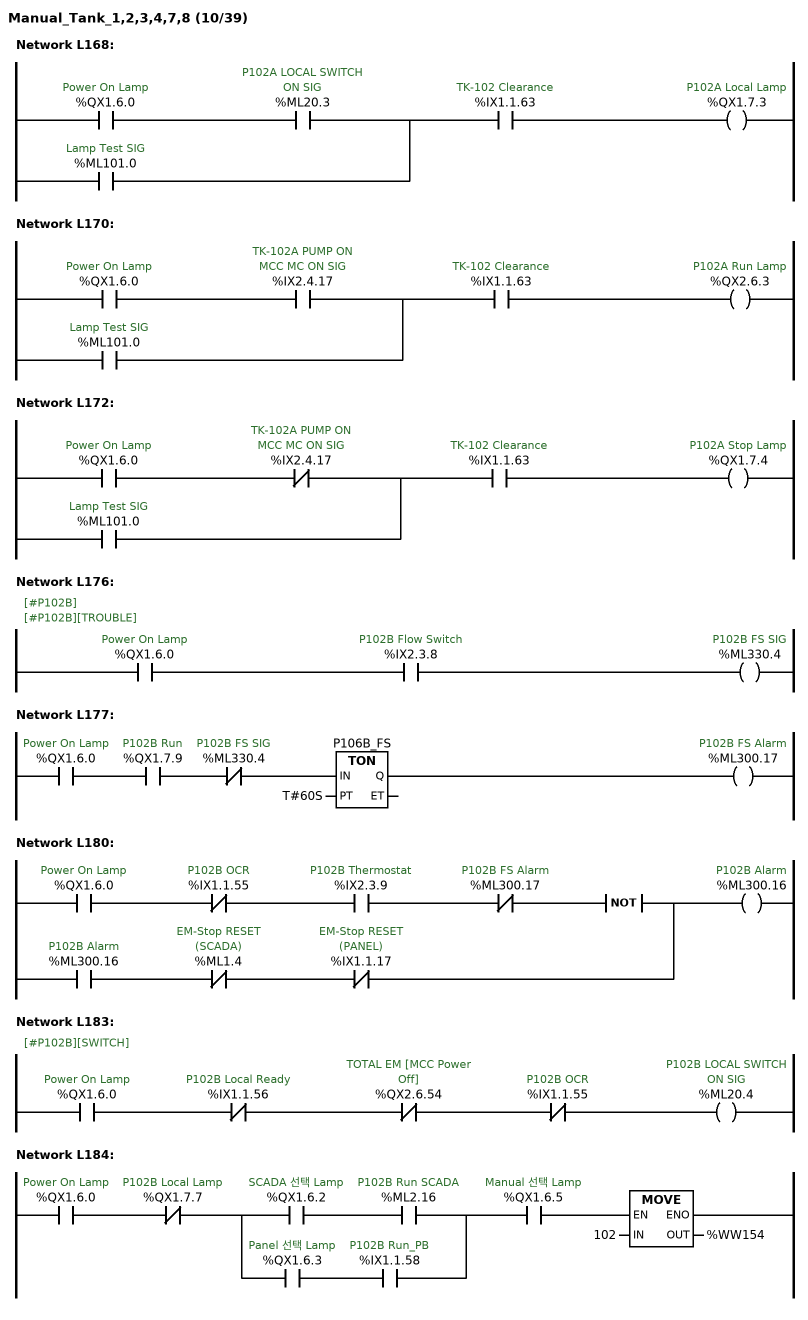
(* [picture p24: Manual_Tank_1,2,3,4,7,8 rungs L168-L184] *)
(* Rung L168 *)
%QX1.7.3 := ((%QX1.6.0 AND %ML20.3) OR %ML101.0) AND %IX1.1.63;
(* Rung L170 *)
%QX2.6.3 := ((%QX1.6.0 AND %IX2.4.17) OR %ML101.0) AND %IX1.1.63;
(* Rung L172 *)
%QX1.7.4 := ((%QX1.6.0 AND NOT %IX2.4.17) OR %ML101.0) AND %IX1.1.63;
(* [#P102B] *)
(* [#P102B][TROUBLE] *)
(* Rung L176 *)
%ML330.4 := %QX1.6.0 AND %IX2.3.8;
(* Rung L177 *)
P106B_FS(IN := %QX1.6.0 AND %QX1.7.9 AND NOT %ML330.4, PT := T#60S);
%ML300.17 := P106B_FS.Q;
(* Rung L180 *)
%ML300.16 := NOT (%QX1.6.0 AND NOT %IX1.1.55 AND %IX2.3.9 AND NOT %ML300.17) OR (%ML300.16 AND NOT %ML1.4 AND NOT %IX1.1.17);
(* [#P102B][SWITCH] *)
(* Rung L183 *)
%ML20.4 := %QX1.6.0 AND NOT %IX1.1.56 AND NOT %QX2.6.54 AND NOT %IX1.1.55;
(* Rung L184 *)
IF %QX1.6.0 AND NOT %QX1.7.7 AND ((%QX1.6.2 AND %ML2.16) OR (%QX1.6.3 AND %IX1.1.58)) AND %QX1.6.5 THEN
    %WW154 := 102;
END_IF;

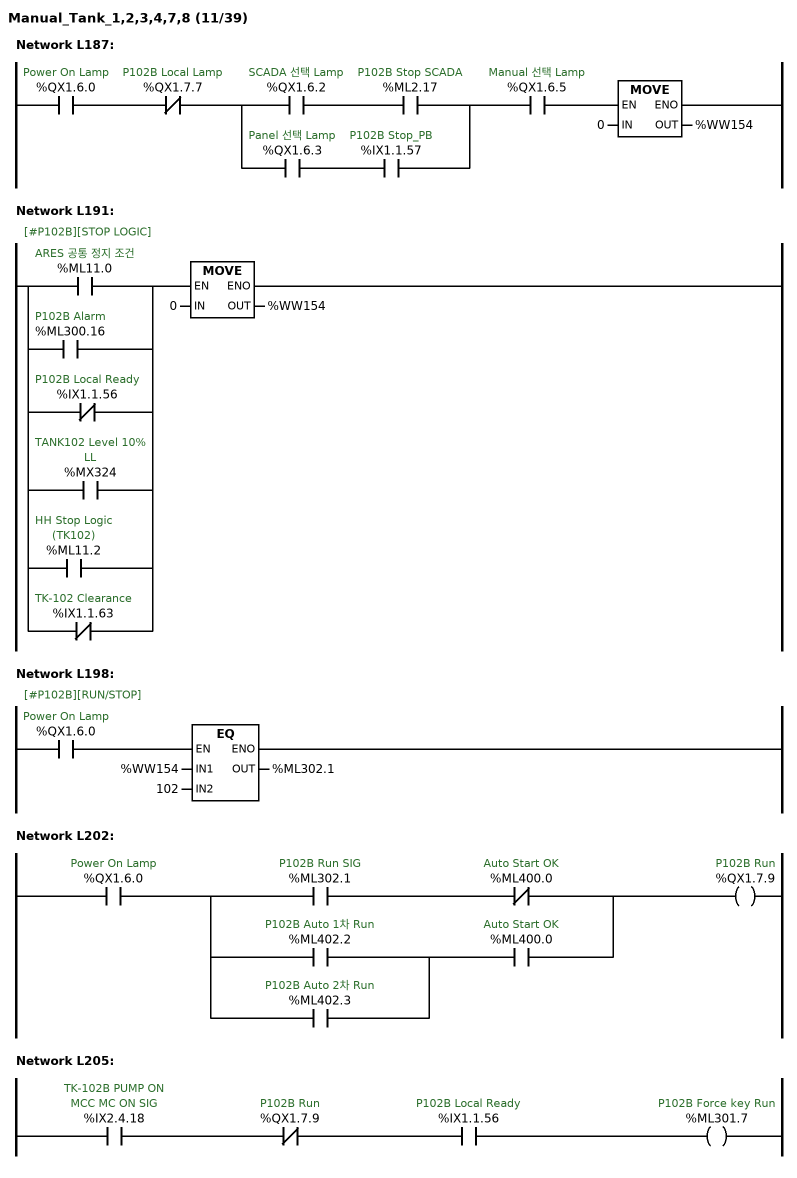
(* Rung L187 *)
IF %QX1.6.0 AND NOT %QX1.7.7 AND ((%QX1.6.2 AND %ML2.17) OR (%QX1.6.3 AND %IX1.1.57)) AND %QX1.6.5 THEN
    %WW154 := 0;
END_IF;
(* [#P102B][STOP LOGIC] *)
(* Rung L191 *)
IF %ML11.0 OR %ML300.16 OR NOT %IX1.1.56 OR %MX324 OR %ML11.2 OR NOT %IX1.1.63 THEN %WW154 := 0; END_IF;
(* [#P102B][RUN/STOP] *)
(* Rung L198 *)
IF %QX1.6.0 THEN %ML302.1 := %WW154 = 102; END_IF;
(* Rung L202 *)
%QX1.7.9 := %QX1.6.0 AND ((%ML302.1 AND NOT %ML400.0) OR ((%ML402.2 OR %ML402.3) AND %ML400.0));
(* Rung L205 *)
%ML301.7 := %IX2.4.18 AND NOT %QX1.7.9 AND %IX1.1.56;

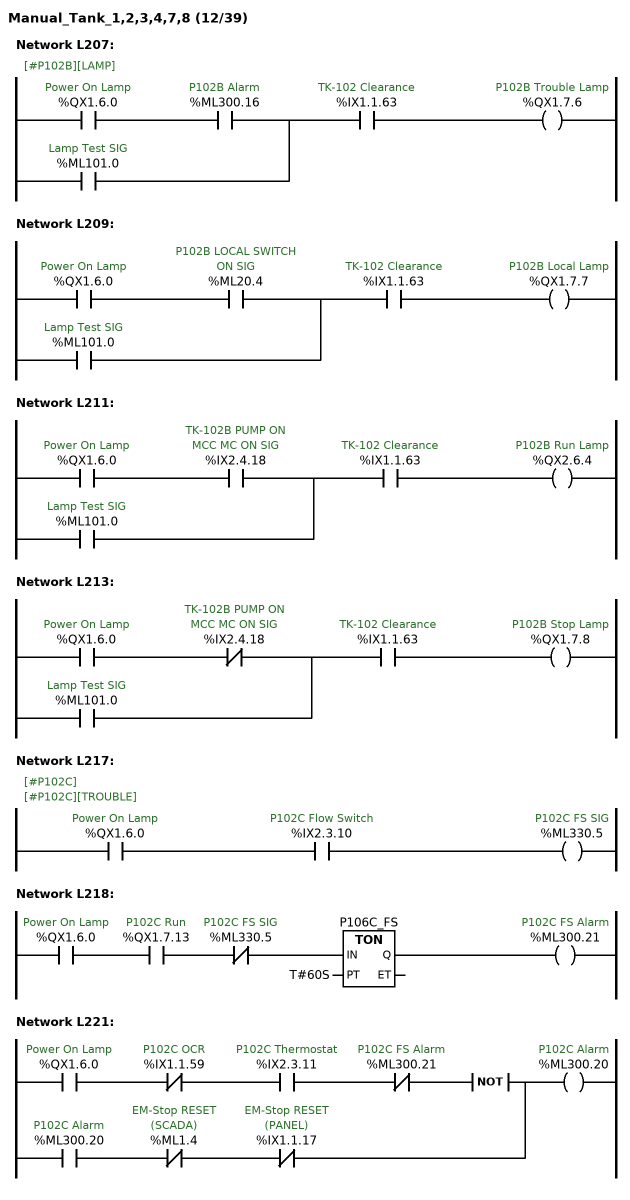
(* [#P102B][LAMP] *)
(* Rung L207 *)
%QX1.7.6 := ((%QX1.6.0 AND %ML300.16) OR %ML101.0) AND %IX1.1.63;
(* Rung L209 *)
%QX1.7.7 := ((%QX1.6.0 AND %ML20.4) OR %ML101.0) AND %IX1.1.63;
(* Rung L211 *)
%QX2.6.4 := ((%QX1.6.0 AND %IX2.4.18) OR %ML101.0) AND %IX1.1.63;
(* Rung L213 *)
%QX1.7.8 := ((%QX1.6.0 AND NOT %IX2.4.18) OR %ML101.0) AND %IX1.1.63;
(* [#P102C] *)
(* [#P102C][TROUBLE] *)
(* Rung L217 *)
%ML330.5 := %QX1.6.0 AND %IX2.3.10;
(* Rung L218 *)
P106C_FS(IN := %QX1.6.0 AND %QX1.7.13 AND NOT %ML330.5, PT := T#60S);
%ML300.21 := P106C_FS.Q;
(* Rung L221 *)
%ML300.20 := NOT (%QX1.6.0 AND NOT %IX1.1.59 AND %IX2.3.11 AND NOT %ML300.21) OR (%ML300.20 AND NOT %ML1.4 AND NOT %IX1.1.17);

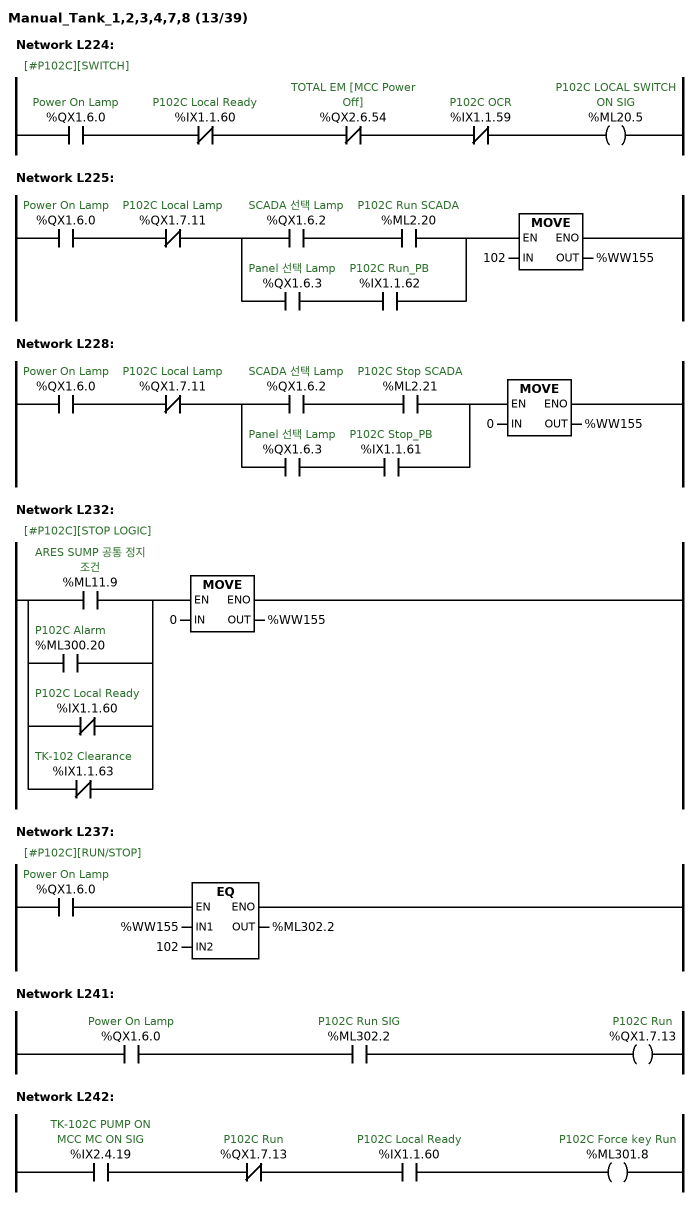
(* [#P102C][SWITCH] *)
(* Rung L224 *)
%ML20.5 := %QX1.6.0 AND NOT %IX1.1.60 AND NOT %QX2.6.54 AND NOT %IX1.1.59;
(* Rung L225 *)
IF %QX1.6.0 AND NOT %QX1.7.11 AND ((%QX1.6.2 AND %ML2.20) OR (%QX1.6.3 AND %IX1.1.62)) THEN
    %WW155 := 102;
END_IF;
(* Rung L228 *)
IF %QX1.6.0 AND NOT %QX1.7.11 AND ((%QX1.6.2 AND %ML2.21) OR (%QX1.6.3 AND %IX1.1.61)) THEN
    %WW155 := 0;
END_IF;
(* [#P102C][STOP LOGIC] *)
(* Rung L232 *)
IF %ML11.9 OR %ML300.20 OR NOT %IX1.1.60 OR NOT %IX1.1.63 THEN %WW155 := 0; END_IF;
(* [#P102C][RUN/STOP] *)
(* Rung L237 *)
IF %QX1.6.0 THEN %ML302.2 := %WW155 = 102; END_IF;
(* Rung L241 *)
%QX1.7.13 := %QX1.6.0 AND %ML302.2;
(* Rung L242 *)
%ML301.8 := %IX2.4.19 AND NOT %QX1.7.13 AND %IX1.1.60;

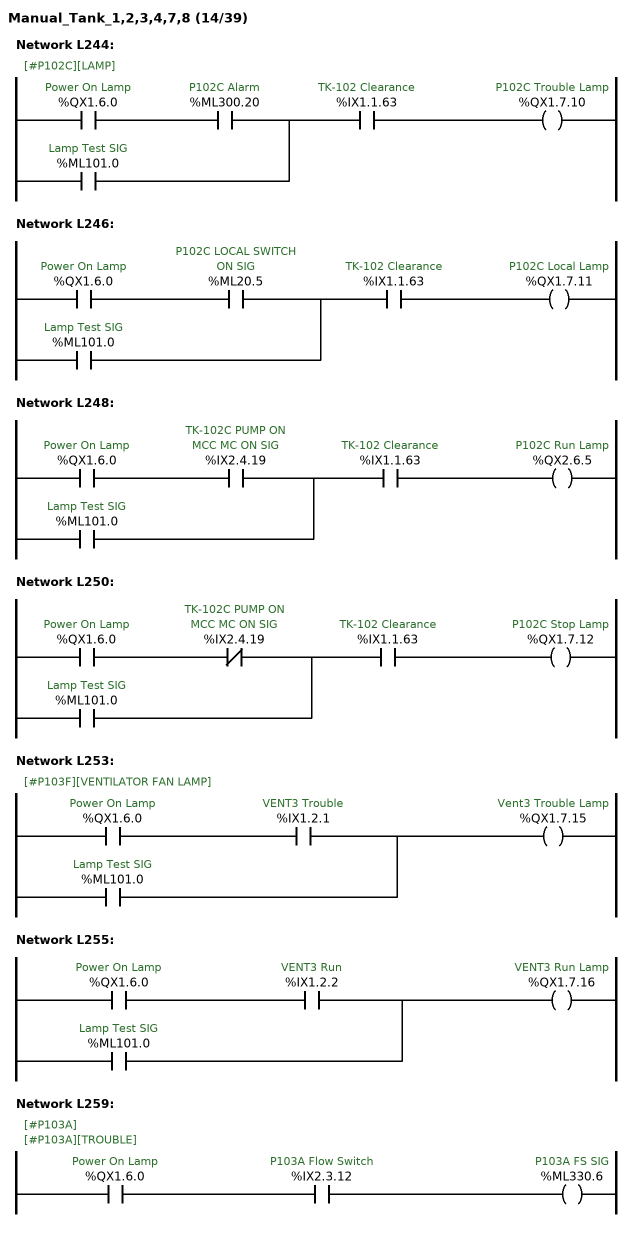
(* [#P102C][LAMP] *)
(* Rung L244 *)
%QX1.7.10 := ((%QX1.6.0 AND %ML300.20) OR %ML101.0) AND %IX1.1.63;
(* Rung L246 *)
%QX1.7.11 := ((%QX1.6.0 AND %ML20.5) OR %ML101.0) AND %IX1.1.63;
(* Rung L248 *)
%QX2.6.5 := ((%QX1.6.0 AND %IX2.4.19) OR %ML101.0) AND %IX1.1.63;
(* Rung L250 *)
%QX1.7.12 := ((%QX1.6.0 AND NOT %IX2.4.19) OR %ML101.0) AND %IX1.1.63;
(* [#P103F][VENTILATOR FAN LAMP] *)
(* Rung L253 *)
%QX1.7.15 := (%QX1.6.0 AND %IX1.2.1) OR %ML101.0;
(* Rung L255 *)
%QX1.7.16 := (%QX1.6.0 AND %IX1.2.2) OR %ML101.0;
(* [#P103A] *)
(* [#P103A][TROUBLE] *)
(* Rung L259 *)
%ML330.6 := %QX1.6.0 AND %IX2.3.12;

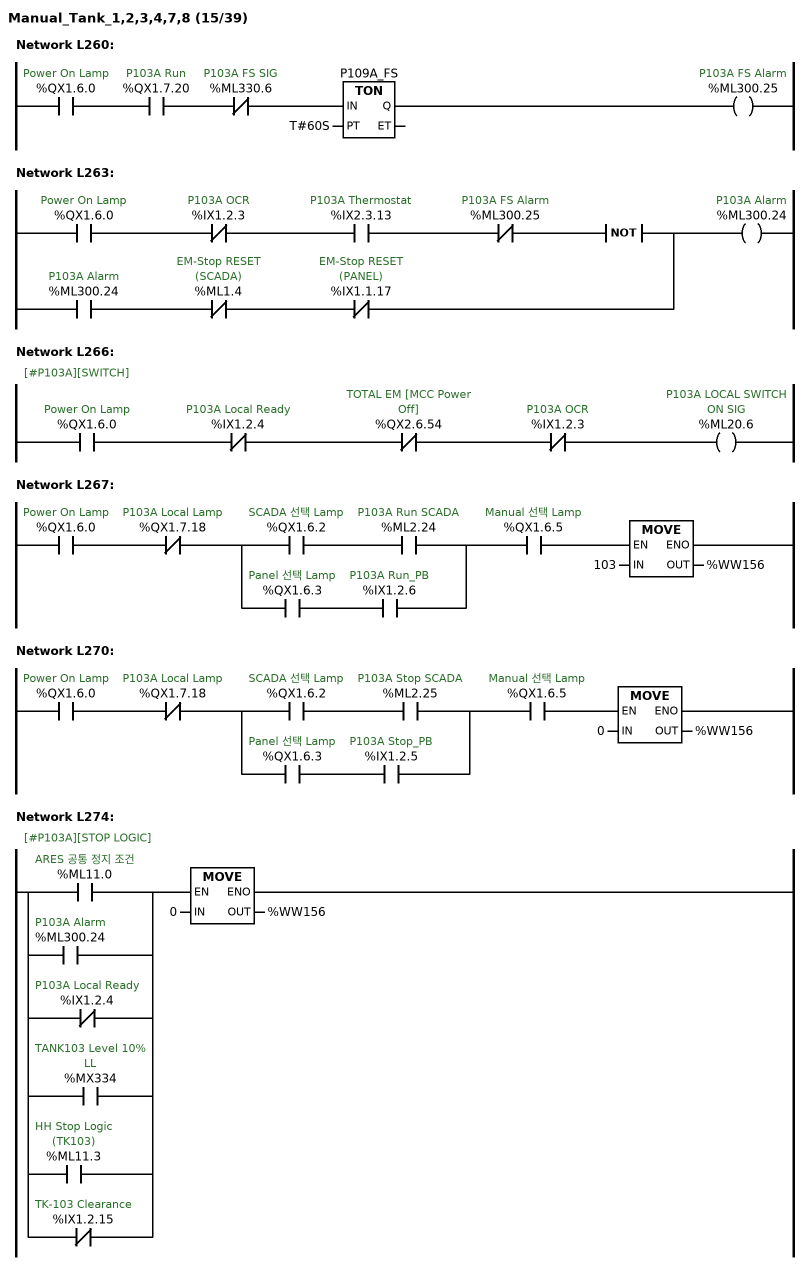
(* Rung L260 *)
P109A_FS(IN := %QX1.6.0 AND %QX1.7.20 AND NOT %ML330.6, PT := T#60S);
%ML300.25 := P109A_FS.Q;
(* Rung L263 *)
%ML300.24 := NOT (%QX1.6.0 AND NOT %IX1.2.3 AND %IX2.3.13 AND NOT %ML300.25) OR (%ML300.24 AND NOT %ML1.4 AND NOT %IX1.1.17);
(* [#P103A][SWITCH] *)
(* Rung L266 *)
%ML20.6 := %QX1.6.0 AND NOT %IX1.2.4 AND NOT %QX2.6.54 AND NOT %IX1.2.3;
(* Rung L267 *)
IF %QX1.6.0 AND NOT %QX1.7.18 AND ((%QX1.6.2 AND %ML2.24) OR (%QX1.6.3 AND %IX1.2.6)) AND %QX1.6.5 THEN
    %WW156 := 103;
END_IF;
(* Rung L270 *)
IF %QX1.6.0 AND NOT %QX1.7.18 AND ((%QX1.6.2 AND %ML2.25) OR (%QX1.6.3 AND %IX1.2.5)) AND %QX1.6.5 THEN
    %WW156 := 0;
END_IF;
(* [#P103A][STOP LOGIC] *)
(* Rung L274 *)
IF %ML11.0 OR %ML300.24 OR NOT %IX1.2.4 OR %MX334 OR %ML11.3 OR NOT %IX1.2.15 THEN %WW156 := 0; END_IF;

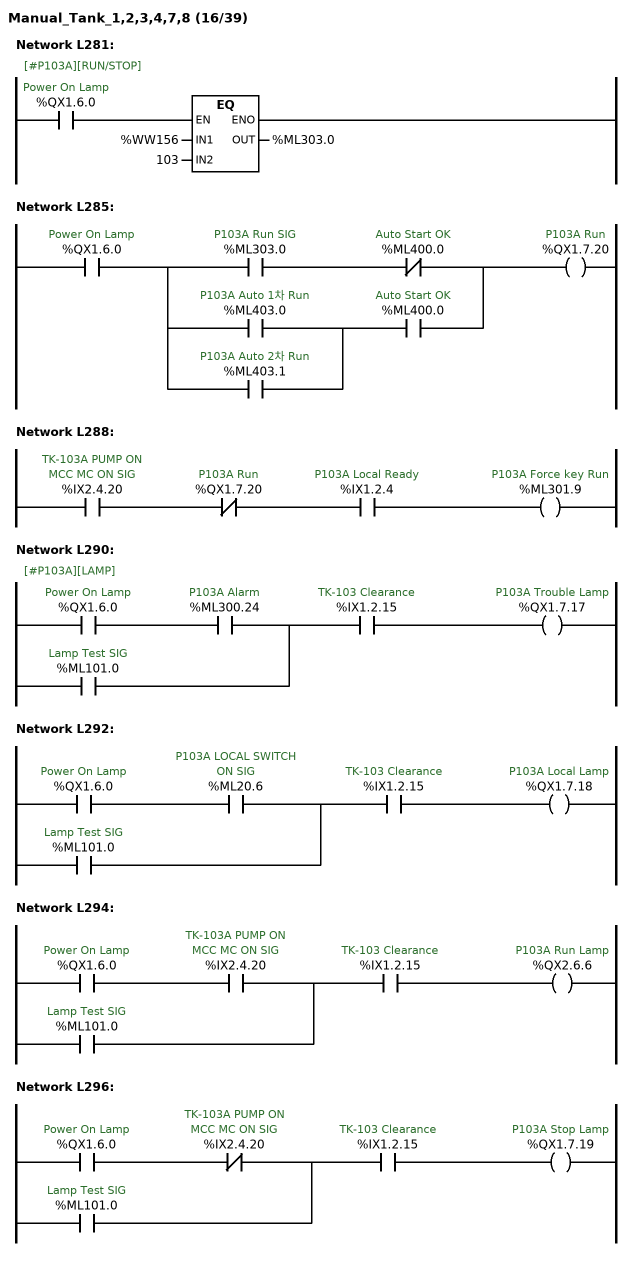
(* [#P103A][RUN/STOP] *)
(* Rung L281 *)
IF %QX1.6.0 THEN %ML303.0 := %WW156 = 103; END_IF;
(* Rung L285 *)
%QX1.7.20 := %QX1.6.0 AND ((%ML303.0 AND NOT %ML400.0) OR ((%ML403.0 OR %ML403.1) AND %ML400.0));
(* Rung L288 *)
%ML301.9 := %IX2.4.20 AND NOT %QX1.7.20 AND %IX1.2.4;
(* [#P103A][LAMP] *)
(* Rung L290 *)
%QX1.7.17 := ((%QX1.6.0 AND %ML300.24) OR %ML101.0) AND %IX1.2.15;
(* Rung L292 *)
%QX1.7.18 := ((%QX1.6.0 AND %ML20.6) OR %ML101.0) AND %IX1.2.15;
(* Rung L294 *)
%QX2.6.6 := ((%QX1.6.0 AND %IX2.4.20) OR %ML101.0) AND %IX1.2.15;
(* Rung L296 *)
%QX1.7.19 := ((%QX1.6.0 AND NOT %IX2.4.20) OR %ML101.0) AND %IX1.2.15;

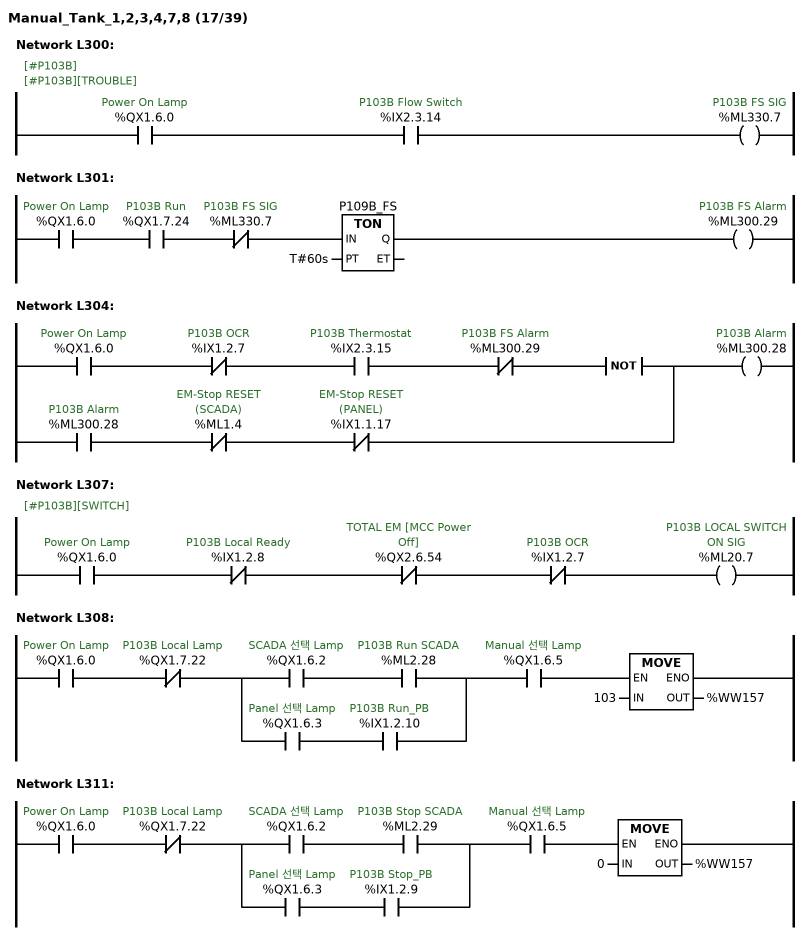
(* [#P103B] *)
(* [#P103B][TROUBLE] *)
(* Rung L300 *)
%ML330.7 := %QX1.6.0 AND %IX2.3.14;
(* Rung L301 *)
P109B_FS(IN := %QX1.6.0 AND %QX1.7.24 AND NOT %ML330.7, PT := T#60s);
%ML300.29 := P109B_FS.Q;
(* Rung L304 *)
%ML300.28 := NOT (%QX1.6.0 AND NOT %IX1.2.7 AND %IX2.3.15 AND NOT %ML300.29) OR (%ML300.28 AND NOT %ML1.4 AND NOT %IX1.1.17);
(* [#P103B][SWITCH] *)
(* Rung L307 *)
%ML20.7 := %QX1.6.0 AND NOT %IX1.2.8 AND NOT %QX2.6.54 AND NOT %IX1.2.7;
(* Rung L308 *)
IF %QX1.6.0 AND NOT %QX1.7.22 AND ((%QX1.6.2 AND %ML2.28) OR (%QX1.6.3 AND %IX1.2.10)) AND %QX1.6.5 THEN
    %WW157 := 103;
END_IF;
(* Rung L311 *)
IF %QX1.6.0 AND NOT %QX1.7.22 AND ((%QX1.6.2 AND %ML2.29) OR (%QX1.6.3 AND %IX1.2.9)) AND %QX1.6.5 THEN
    %WW157 := 0;
END_IF;

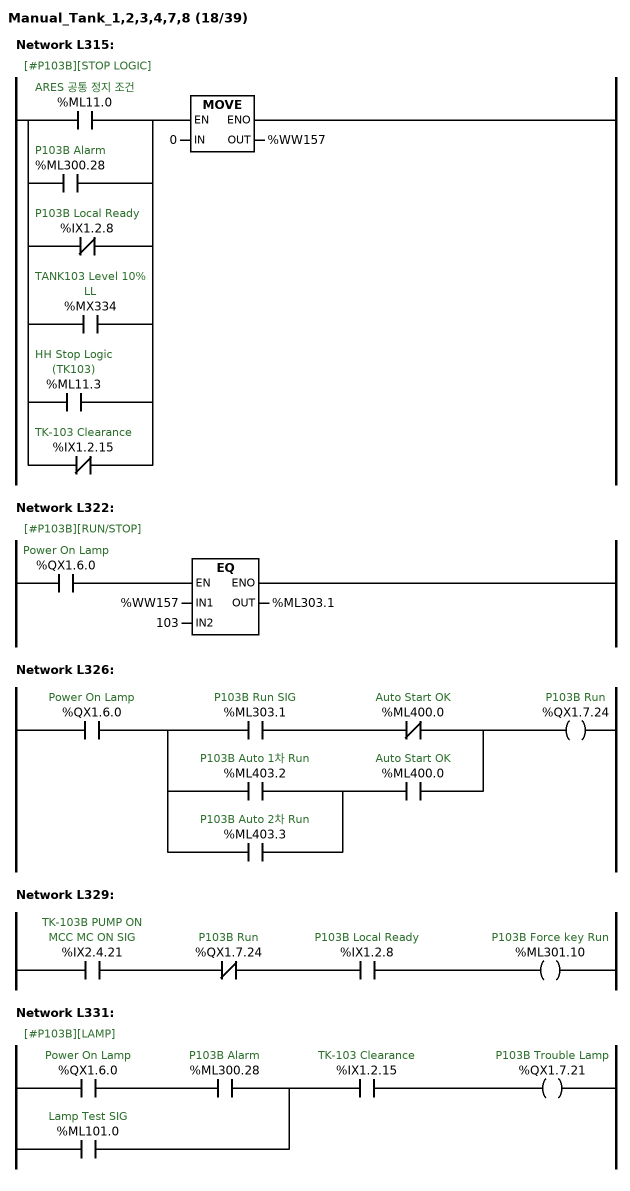
(* [#P103B][STOP LOGIC] *)
(* Rung L315 *)
IF %ML11.0 OR %ML300.28 OR NOT %IX1.2.8 OR %MX334 OR %ML11.3 OR NOT %IX1.2.15 THEN %WW157 := 0; END_IF;
(* [#P103B][RUN/STOP] *)
(* Rung L322 *)
IF %QX1.6.0 THEN %ML303.1 := %WW157 = 103; END_IF;
(* Rung L326 *)
%QX1.7.24 := %QX1.6.0 AND ((%ML303.1 AND NOT %ML400.0) OR ((%ML403.2 OR %ML403.3) AND %ML400.0));
(* Rung L329 *)
%ML301.10 := %IX2.4.21 AND NOT %QX1.7.24 AND %IX1.2.8;
(* [#P103B][LAMP] *)
(* Rung L331 *)
%QX1.7.21 := ((%QX1.6.0 AND %ML300.28) OR %ML101.0) AND %IX1.2.15;

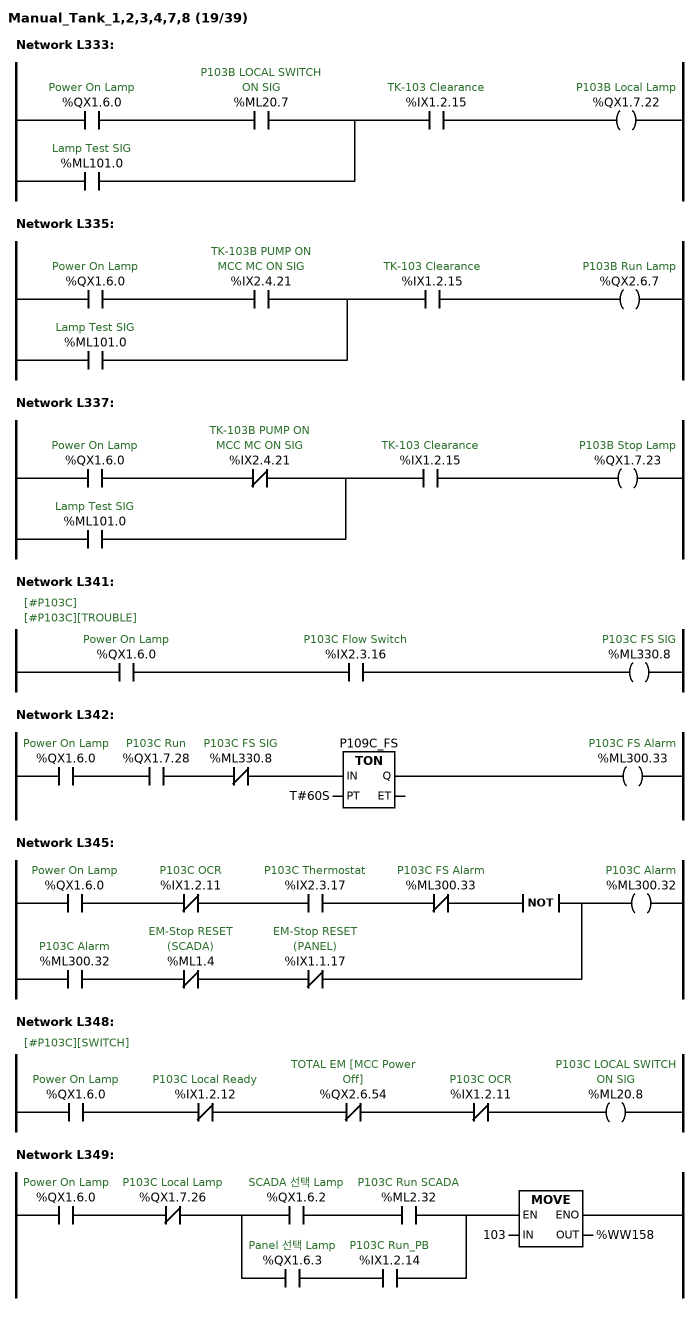
(* Rung L333 *)
%QX1.7.22 := ((%QX1.6.0 AND %ML20.7) OR %ML101.0) AND %IX1.2.15;
(* Rung L335 *)
%QX2.6.7 := ((%QX1.6.0 AND %IX2.4.21) OR %ML101.0) AND %IX1.2.15;
(* Rung L337 *)
%QX1.7.23 := ((%QX1.6.0 AND NOT %IX2.4.21) OR %ML101.0) AND %IX1.2.15;
(* [#P103C] *)
(* [#P103C][TROUBLE] *)
(* Rung L341 *)
%ML330.8 := %QX1.6.0 AND %IX2.3.16;
(* Rung L342 *)
P109C_FS(IN := %QX1.6.0 AND %QX1.7.28 AND NOT %ML330.8, PT := T#60S);
%ML300.33 := P109C_FS.Q;
(* Rung L345 *)
%ML300.32 := NOT (%QX1.6.0 AND NOT %IX1.2.11 AND %IX2.3.17 AND NOT %ML300.33) OR (%ML300.32 AND NOT %ML1.4 AND NOT %IX1.1.17);
(* [#P103C][SWITCH] *)
(* Rung L348 *)
%ML20.8 := %QX1.6.0 AND NOT %IX1.2.12 AND NOT %QX2.6.54 AND NOT %IX1.2.11;
(* Rung L349 *)
IF %QX1.6.0 AND NOT %QX1.7.26 AND ((%QX1.6.2 AND %ML2.32) OR (%QX1.6.3 AND %IX1.2.14)) THEN
    %WW158 := 103;
END_IF;

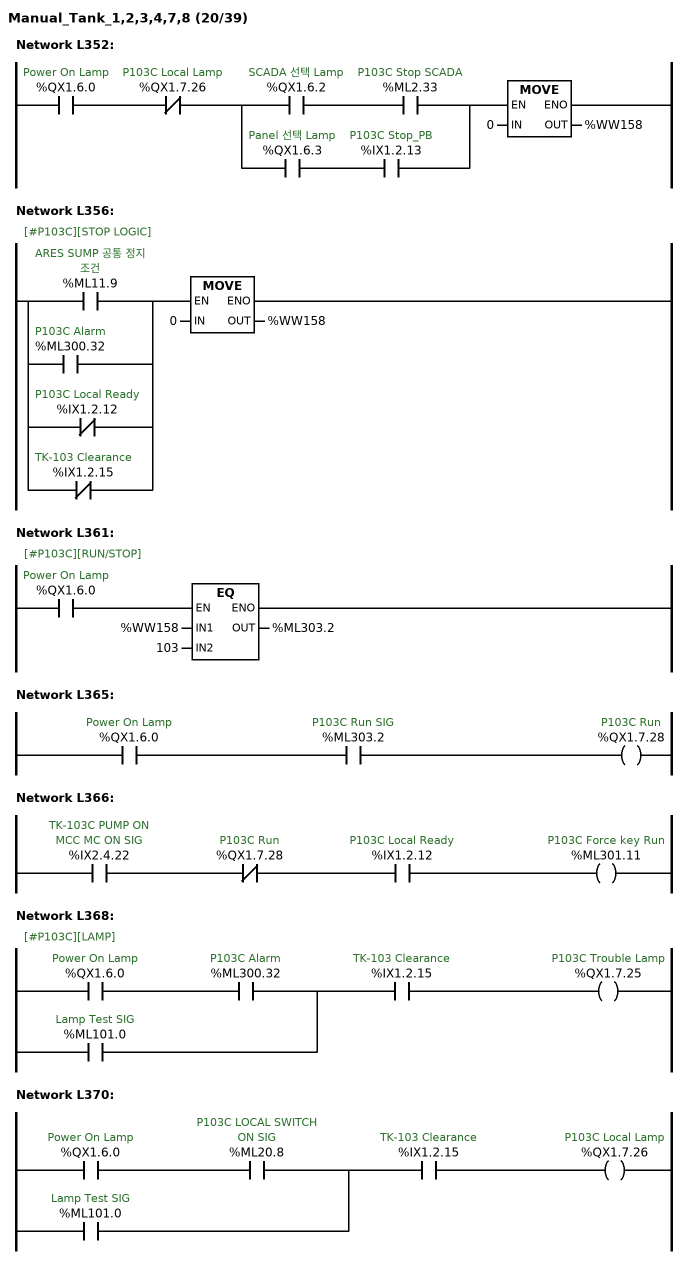
(* Rung L352 *)
IF %QX1.6.0 AND NOT %QX1.7.26 AND ((%QX1.6.2 AND %ML2.33) OR (%QX1.6.3 AND %IX1.2.13)) THEN
    %WW158 := 0;
END_IF;
(* [#P103C][STOP LOGIC] *)
(* Rung L356 *)
IF %ML11.9 OR %ML300.32 OR NOT %IX1.2.12 OR NOT %IX1.2.15 THEN %WW158 := 0; END_IF;
(* [#P103C][RUN/STOP] *)
(* Rung L361 *)
IF %QX1.6.0 THEN %ML303.2 := %WW158 = 103; END_IF;
(* Rung L365 *)
%QX1.7.28 := %QX1.6.0 AND %ML303.2;
(* Rung L366 *)
%ML301.11 := %IX2.4.22 AND NOT %QX1.7.28 AND %IX1.2.12;
(* [#P103C][LAMP] *)
(* Rung L368 *)
%QX1.7.25 := ((%QX1.6.0 AND %ML300.32) OR %ML101.0) AND %IX1.2.15;
(* Rung L370 *)
%QX1.7.26 := ((%QX1.6.0 AND %ML20.8) OR %ML101.0) AND %IX1.2.15;

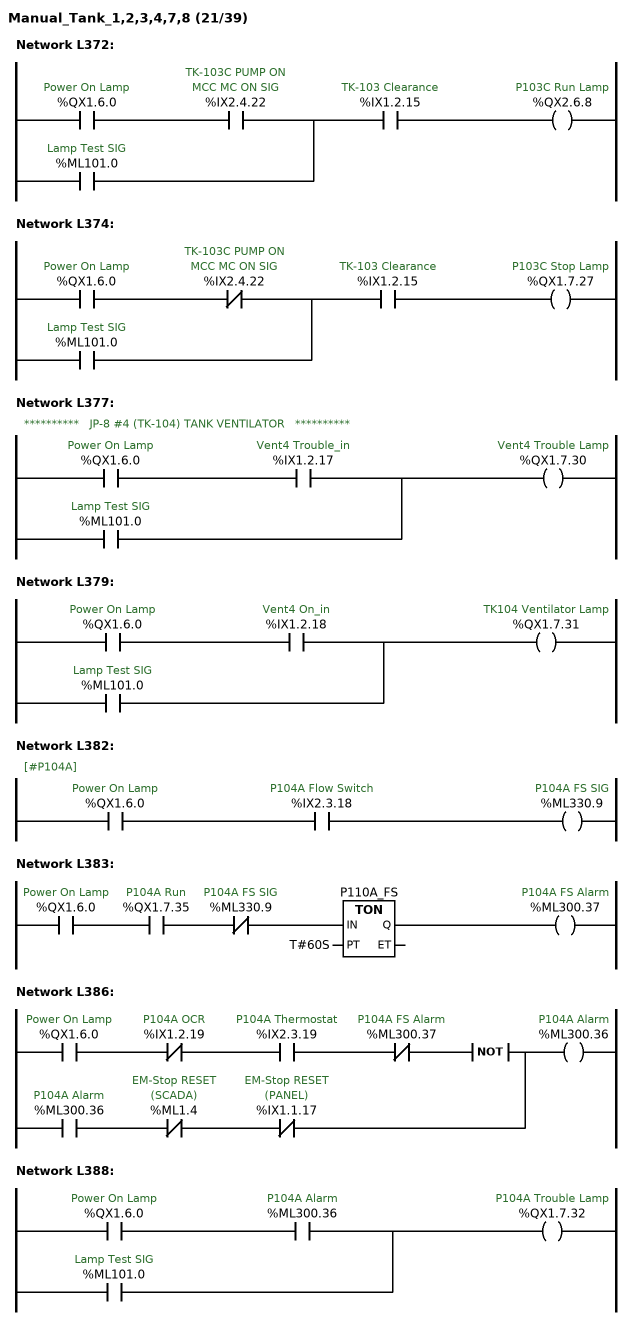
(* Rung L372 *)
%QX2.6.8 := ((%QX1.6.0 AND %IX2.4.22) OR %ML101.0) AND %IX1.2.15;
(* Rung L374 *)
%QX1.7.27 := ((%QX1.6.0 AND NOT %IX2.4.22) OR %ML101.0) AND %IX1.2.15;
(* **********   JP-8 #4 (TK-104) TANK VENTILATOR   ********** *)
(* Rung L377 *)
%QX1.7.30 := (%QX1.6.0 AND %IX1.2.17) OR %ML101.0;
(* Rung L379 *)
%QX1.7.31 := (%QX1.6.0 AND %IX1.2.18) OR %ML101.0;
(* [#P104A] *)
(* Rung L382 *)
%ML330.9 := %QX1.6.0 AND %IX2.3.18;
(* Rung L383 *)
P110A_FS(IN := %QX1.6.0 AND %QX1.7.35 AND NOT %ML330.9, PT := T#60S);
%ML300.37 := P110A_FS.Q;
(* Rung L386 *)
%ML300.36 := NOT (%QX1.6.0 AND NOT %IX1.2.19 AND %IX2.3.19 AND NOT %ML300.37) OR (%ML300.36 AND NOT %ML1.4 AND NOT %IX1.1.17);
(* Rung L388 *)
%QX1.7.32 := (%QX1.6.0 AND %ML300.36) OR %ML101.0;

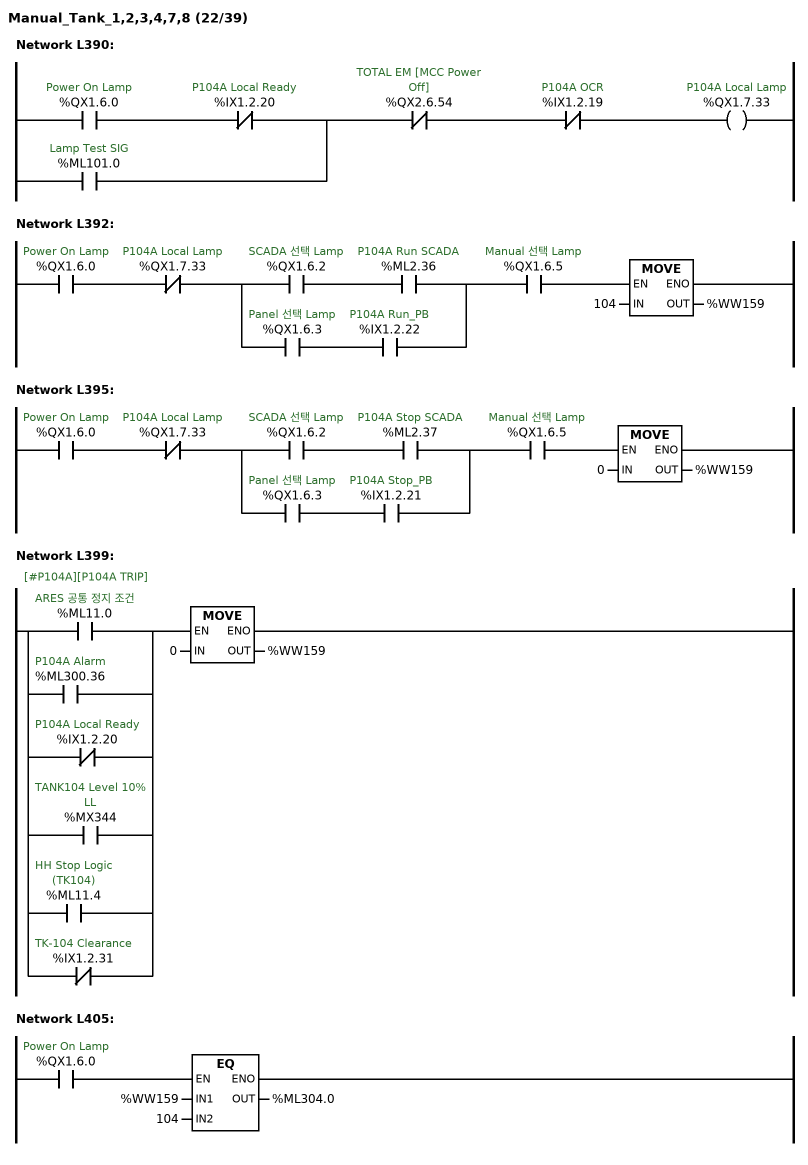
(* Rung L390 *)
%QX1.7.33 := ((%QX1.6.0 AND NOT %IX1.2.20) OR %ML101.0) AND NOT %QX2.6.54 AND NOT %IX1.2.19;
(* Rung L392 *)
IF %QX1.6.0 AND NOT %QX1.7.33 AND ((%QX1.6.2 AND %ML2.36) OR (%QX1.6.3 AND %IX1.2.22)) AND %QX1.6.5 THEN
    %WW159 := 104;
END_IF;
(* Rung L395 *)
IF %QX1.6.0 AND NOT %QX1.7.33 AND ((%QX1.6.2 AND %ML2.37) OR (%QX1.6.3 AND %IX1.2.21)) AND %QX1.6.5 THEN
    %WW159 := 0;
END_IF;
(* [#P104A][P104A TRIP] *)
(* Rung L399 *)
IF %ML11.0 OR %ML300.36 OR NOT %IX1.2.20 OR %MX344 OR %ML11.4 OR NOT %IX1.2.31 THEN %WW159 := 0; END_IF;
(* Rung L405 *)
IF %QX1.6.0 THEN %ML304.0 := %WW159 = 104; END_IF;

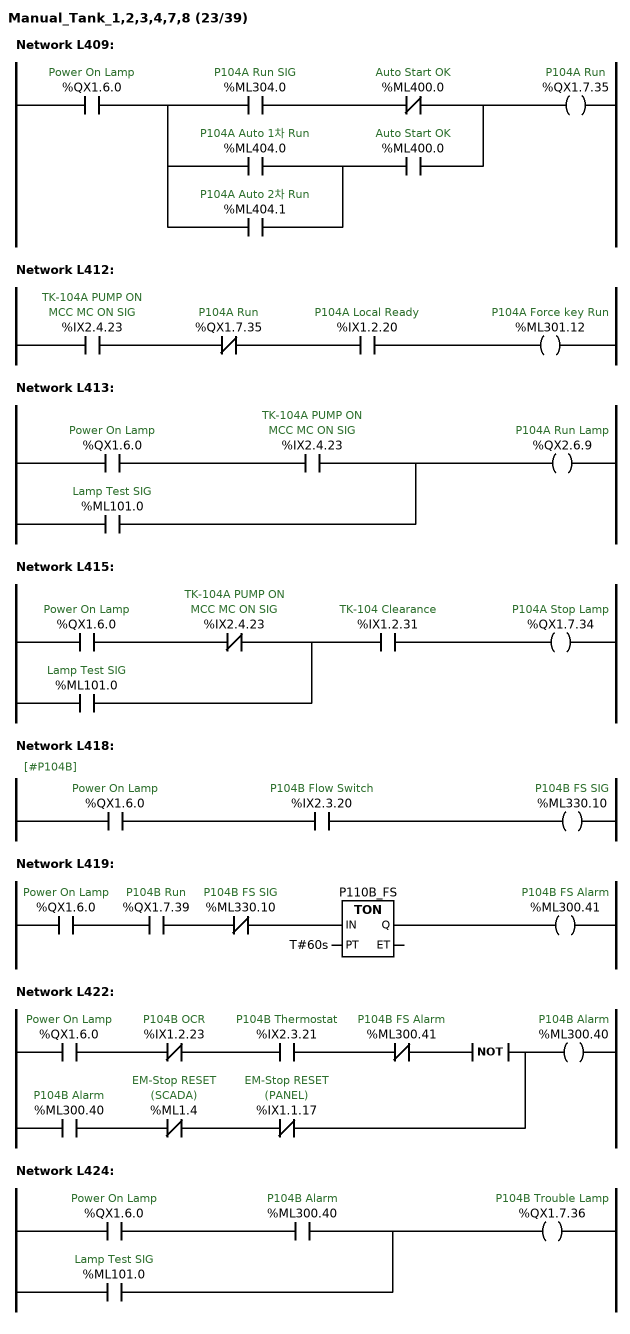
(* Rung L409 *)
%QX1.7.35 := %QX1.6.0 AND ((%ML304.0 AND NOT %ML400.0) OR ((%ML404.0 OR %ML404.1) AND %ML400.0));
(* Rung L412 *)
%ML301.12 := %IX2.4.23 AND NOT %QX1.7.35 AND %IX1.2.20;
(* Rung L413 *)
%QX2.6.9 := (%QX1.6.0 AND %IX2.4.23) OR %ML101.0;
(* Rung L415 *)
%QX1.7.34 := ((%QX1.6.0 AND NOT %IX2.4.23) OR %ML101.0) AND %IX1.2.31;
(* [#P104B] *)
(* Rung L418 *)
%ML330.10 := %QX1.6.0 AND %IX2.3.20;
(* Rung L419 *)
P110B_FS(IN := %QX1.6.0 AND %QX1.7.39 AND NOT %ML330.10, PT := T#60s);
%ML300.41 := P110B_FS.Q;
(* Rung L422 *)
%ML300.40 := NOT (%QX1.6.0 AND NOT %IX1.2.23 AND %IX2.3.21 AND NOT %ML300.41) OR (%ML300.40 AND NOT %ML1.4 AND NOT %IX1.1.17);
(* Rung L424 *)
%QX1.7.36 := (%QX1.6.0 AND %ML300.40) OR %ML101.0;

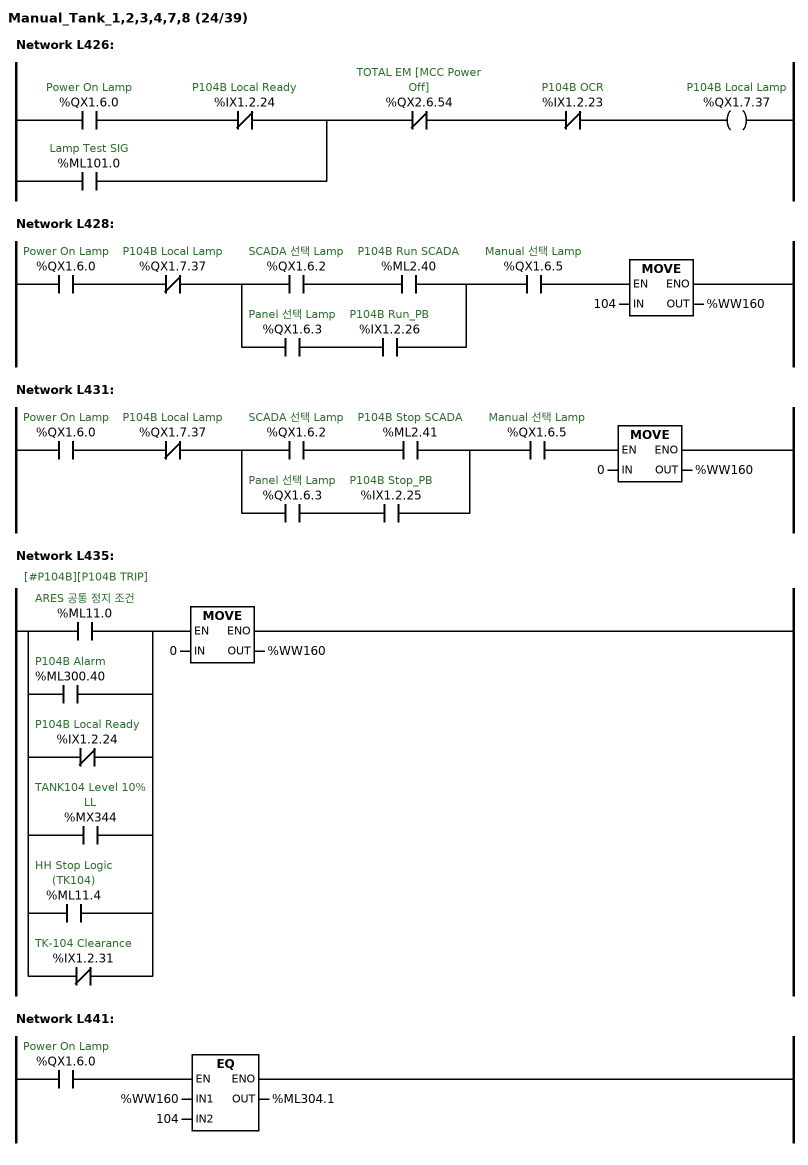
(* Rung L426 *)
%QX1.7.37 := ((%QX1.6.0 AND NOT %IX1.2.24) OR %ML101.0) AND NOT %QX2.6.54 AND NOT %IX1.2.23;
(* Rung L428 *)
IF %QX1.6.0 AND NOT %QX1.7.37 AND ((%QX1.6.2 AND %ML2.40) OR (%QX1.6.3 AND %IX1.2.26)) AND %QX1.6.5 THEN
    %WW160 := 104;
END_IF;
(* Rung L431 *)
IF %QX1.6.0 AND NOT %QX1.7.37 AND ((%QX1.6.2 AND %ML2.41) OR (%QX1.6.3 AND %IX1.2.25)) AND %QX1.6.5 THEN
    %WW160 := 0;
END_IF;
(* [#P104B][P104B TRIP] *)
(* Rung L435 *)
IF %ML11.0 OR %ML300.40 OR NOT %IX1.2.24 OR %MX344 OR %ML11.4 OR NOT %IX1.2.31 THEN %WW160 := 0; END_IF;
(* Rung L441 *)
IF %QX1.6.0 THEN %ML304.1 := %WW160 = 104; END_IF;

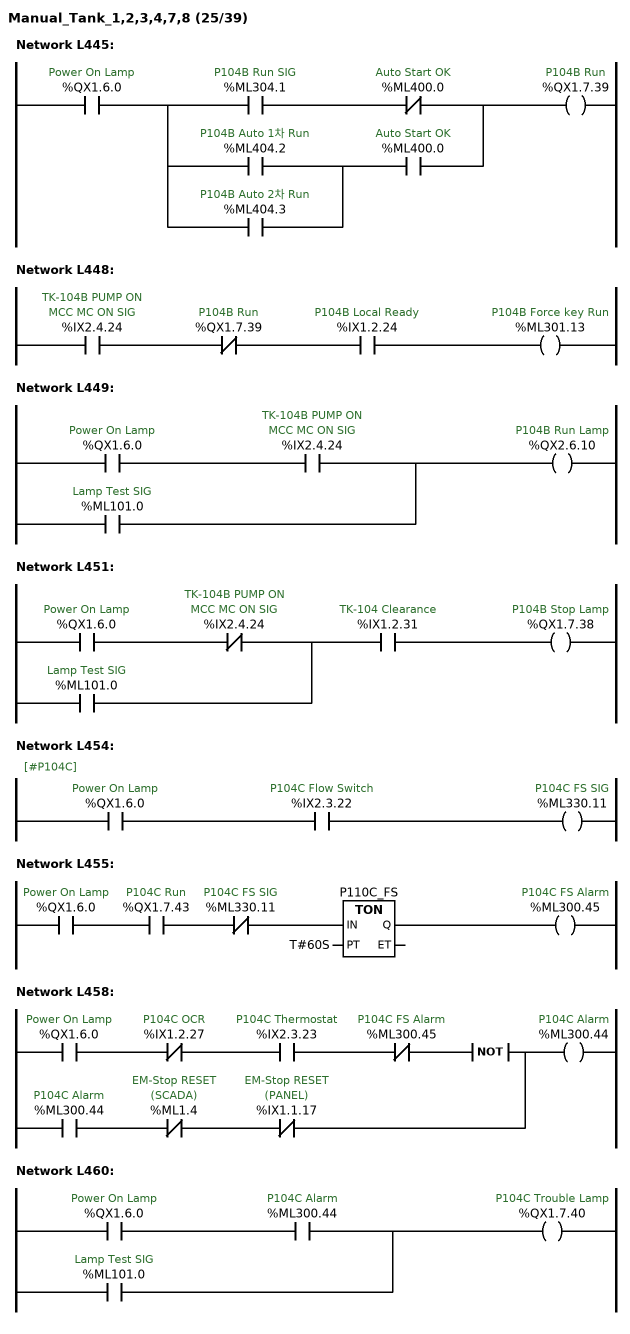
(* Rung L445 *)
%QX1.7.39 := %QX1.6.0 AND ((%ML304.1 AND NOT %ML400.0) OR ((%ML404.2 OR %ML404.3) AND %ML400.0));
(* Rung L448 *)
%ML301.13 := %IX2.4.24 AND NOT %QX1.7.39 AND %IX1.2.24;
(* Rung L449 *)
%QX2.6.10 := (%QX1.6.0 AND %IX2.4.24) OR %ML101.0;
(* Rung L451 *)
%QX1.7.38 := ((%QX1.6.0 AND NOT %IX2.4.24) OR %ML101.0) AND %IX1.2.31;
(* [#P104C] *)
(* Rung L454 *)
%ML330.11 := %QX1.6.0 AND %IX2.3.22;
(* Rung L455 *)
P110C_FS(IN := %QX1.6.0 AND %QX1.7.43 AND NOT %ML330.11, PT := T#60S);
%ML300.45 := P110C_FS.Q;
(* Rung L458 *)
%ML300.44 := NOT (%QX1.6.0 AND NOT %IX1.2.27 AND %IX2.3.23 AND NOT %ML300.45) OR (%ML300.44 AND NOT %ML1.4 AND NOT %IX1.1.17);
(* Rung L460 *)
%QX1.7.40 := (%QX1.6.0 AND %ML300.44) OR %ML101.0;

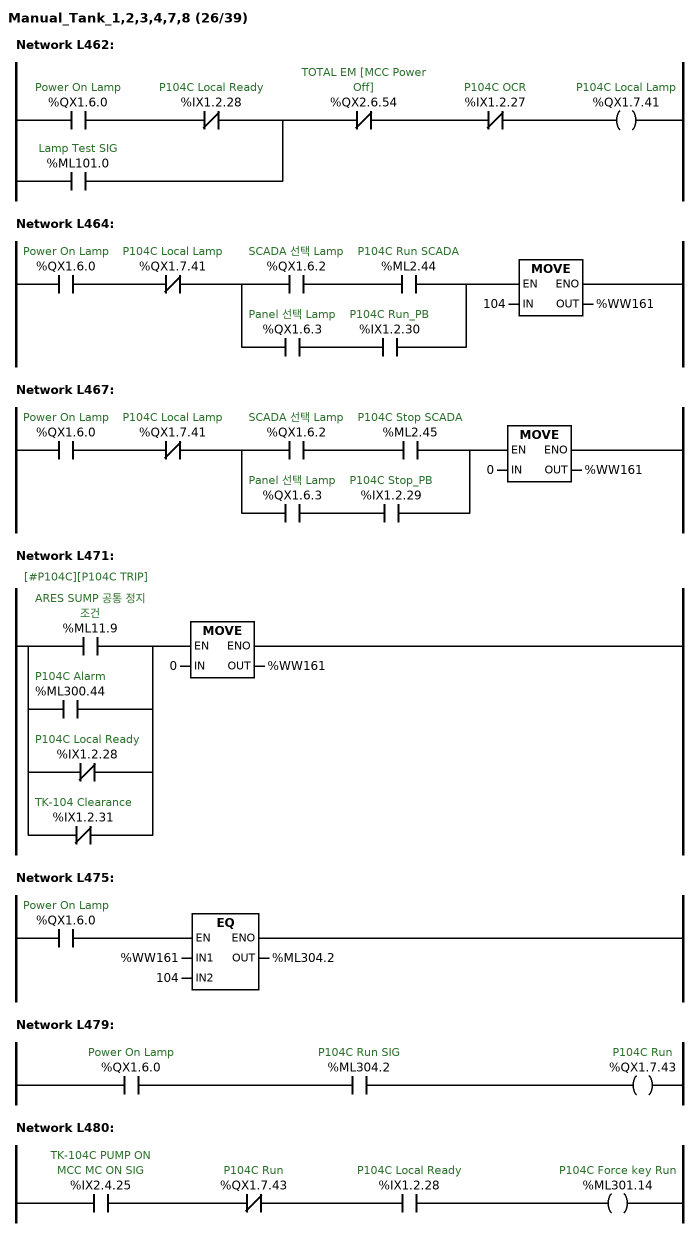
(* Rung L462 *)
%QX1.7.41 := ((%QX1.6.0 AND NOT %IX1.2.28) OR %ML101.0) AND NOT %QX2.6.54 AND NOT %IX1.2.27;
(* Rung L464 *)
IF %QX1.6.0 AND NOT %QX1.7.41 AND ((%QX1.6.2 AND %ML2.44) OR (%QX1.6.3 AND %IX1.2.30)) THEN
    %WW161 := 104;
END_IF;
(* Rung L467 *)
IF %QX1.6.0 AND NOT %QX1.7.41 AND ((%QX1.6.2 AND %ML2.45) OR (%QX1.6.3 AND %IX1.2.29)) THEN
    %WW161 := 0;
END_IF;
(* [#P104C][P104C TRIP] *)
(* Rung L471 *)
IF %ML11.9 OR %ML300.44 OR NOT %IX1.2.28 OR NOT %IX1.2.31 THEN %WW161 := 0; END_IF;
(* Rung L475 *)
IF %QX1.6.0 THEN %ML304.2 := %WW161 = 104; END_IF;
(* Rung L479 *)
%QX1.7.43 := %QX1.6.0 AND %ML304.2;
(* Rung L480 *)
%ML301.14 := %IX2.4.25 AND NOT %QX1.7.43 AND %IX1.2.28;

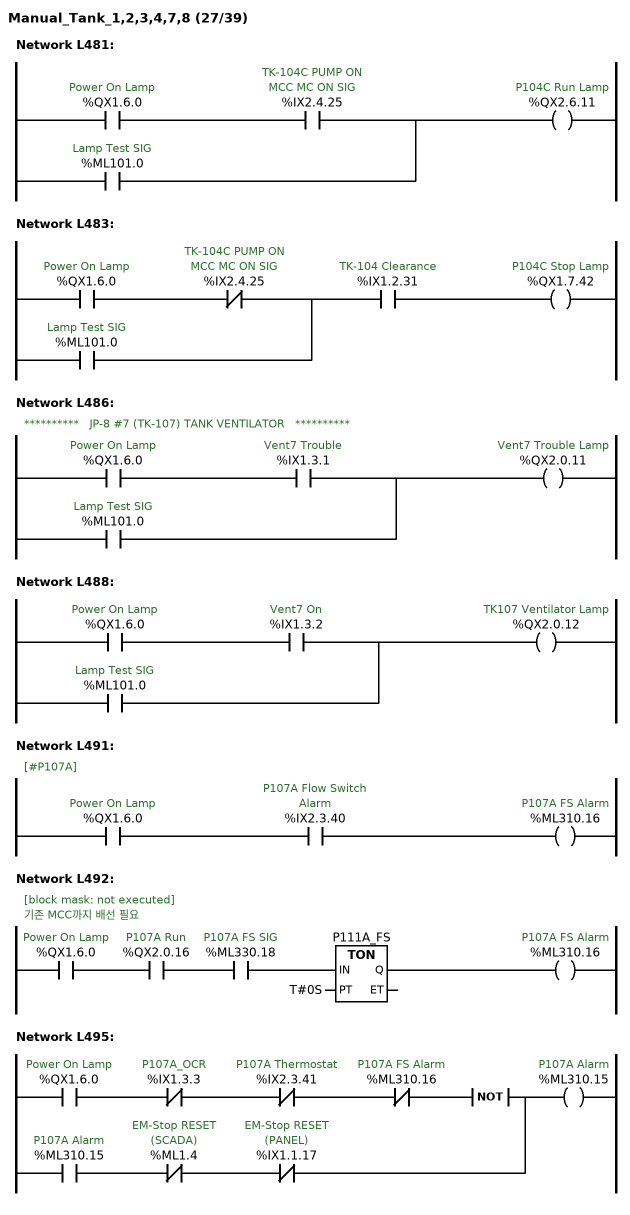
(* Rung L481 *)
%QX2.6.11 := (%QX1.6.0 AND %IX2.4.25) OR %ML101.0;
(* Rung L483 *)
%QX1.7.42 := ((%QX1.6.0 AND NOT %IX2.4.25) OR %ML101.0) AND %IX1.2.31;
(* **********   JP-8 #7 (TK-107) TANK VENTILATOR   ********** *)
(* Rung L486 *)
%QX2.0.11 := (%QX1.6.0 AND %IX1.3.1) OR %ML101.0;
(* Rung L488 *)
%QX2.0.12 := (%QX1.6.0 AND %IX1.3.2) OR %ML101.0;
(* [#P107A] *)
(* Rung L491 *)
%ML310.16 := %QX1.6.0 AND %IX2.3.40;
(* Rung L492 is block-masked: not executed *)
// P111A_FS(IN := %QX1.6.0 AND %QX2.0.16 AND %ML330.18, PT := T#0S);
// %ML310.16 := P111A_FS.Q;
(* 기존 MCC까지 배선 필요 *)
(* Rung L495 *)
%ML310.15 := NOT (%QX1.6.0 AND NOT %IX1.3.3 AND NOT %IX2.3.41 AND NOT %ML310.16) OR (%ML310.15 AND NOT %ML1.4 AND NOT %IX1.1.17);

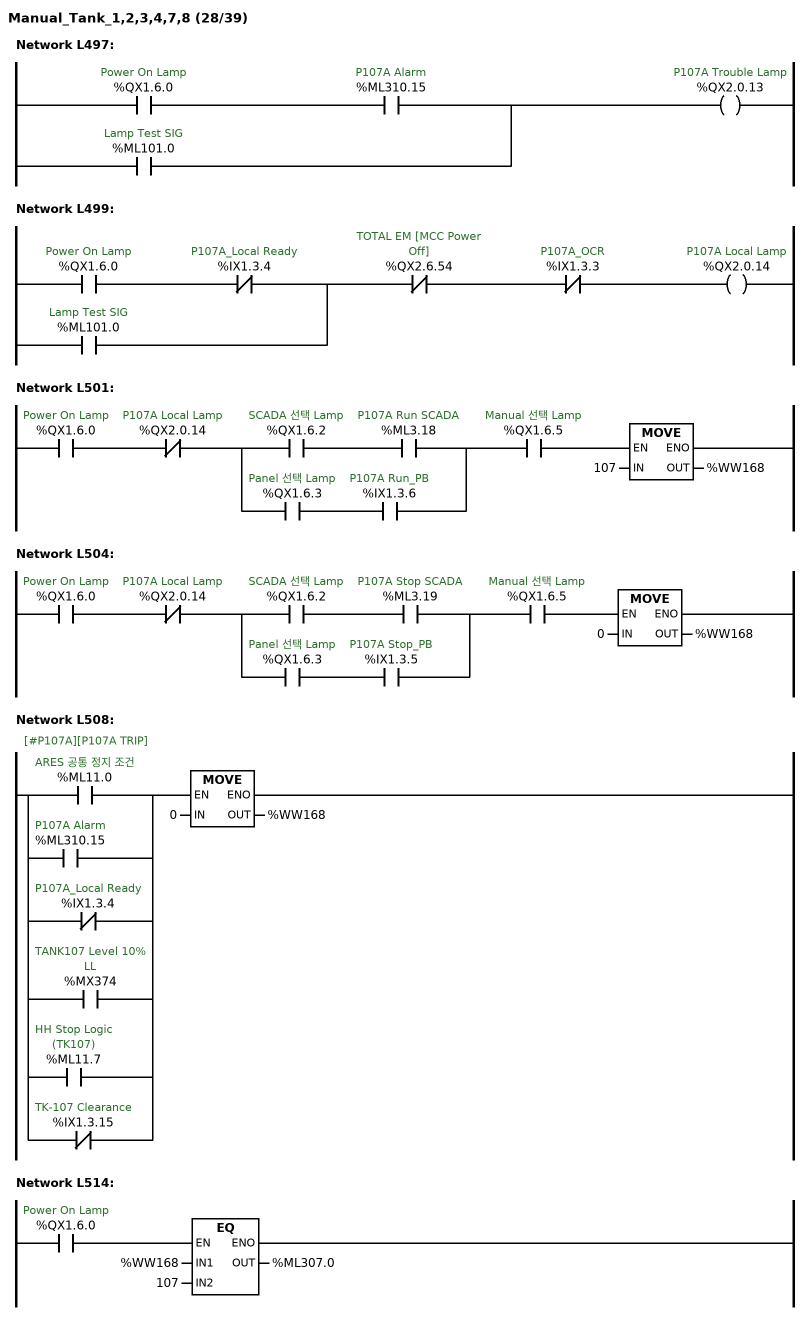
(* Rung L497 *)
%QX2.0.13 := (%QX1.6.0 AND %ML310.15) OR %ML101.0;
(* Rung L499 *)
%QX2.0.14 := ((%QX1.6.0 AND NOT %IX1.3.4) OR %ML101.0) AND NOT %QX2.6.54 AND NOT %IX1.3.3;
(* Rung L501 *)
IF %QX1.6.0 AND NOT %QX2.0.14 AND ((%QX1.6.2 AND %ML3.18) OR (%QX1.6.3 AND %IX1.3.6)) AND %QX1.6.5 THEN
    %WW168 := 107;
END_IF;
(* Rung L504 *)
IF %QX1.6.0 AND NOT %QX2.0.14 AND ((%QX1.6.2 AND %ML3.19) OR (%QX1.6.3 AND %IX1.3.5)) AND %QX1.6.5 THEN
    %WW168 := 0;
END_IF;
(* [#P107A][P107A TRIP] *)
(* Rung L508 *)
IF %ML11.0 OR %ML310.15 OR NOT %IX1.3.4 OR %MX374 OR %ML11.7 OR NOT %IX1.3.15 THEN %WW168 := 0; END_IF;
(* Rung L514 *)
IF %QX1.6.0 THEN %ML307.0 := %WW168 = 107; END_IF;

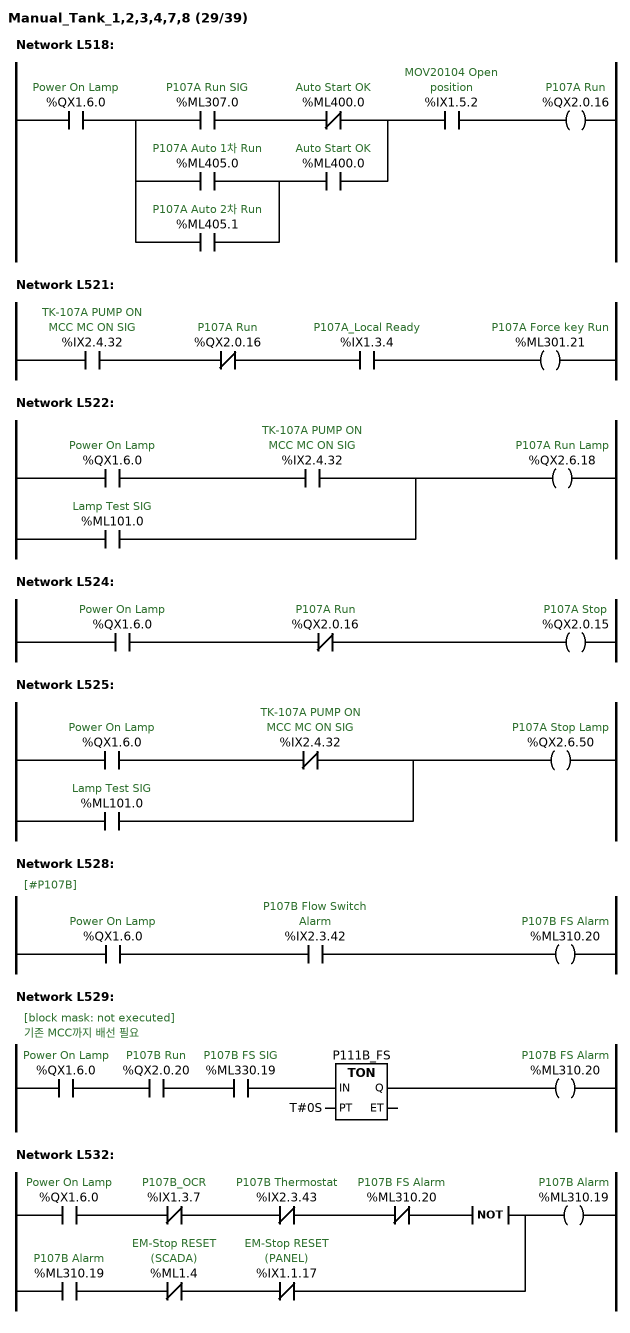
(* Rung L518 *)
%QX2.0.16 := %QX1.6.0 AND ((%ML307.0 AND NOT %ML400.0) OR ((%ML405.0 OR %ML405.1) AND %ML400.0)) AND %IX1.5.2;
(* Rung L521 *)
%ML301.21 := %IX2.4.32 AND NOT %QX2.0.16 AND %IX1.3.4;
(* Rung L522 *)
%QX2.6.18 := (%QX1.6.0 AND %IX2.4.32) OR %ML101.0;
(* Rung L524 *)
%QX2.0.15 := %QX1.6.0 AND NOT %QX2.0.16;
(* Rung L525 *)
%QX2.6.50 := (%QX1.6.0 AND NOT %IX2.4.32) OR %ML101.0;
(* [#P107B] *)
(* Rung L528 *)
%ML310.20 := %QX1.6.0 AND %IX2.3.42;
(* Rung L529 is block-masked: not executed *)
// P111B_FS(IN := %QX1.6.0 AND %QX2.0.20 AND %ML330.19, PT := T#0S);
// %ML310.20 := P111B_FS.Q;
(* 기존 MCC까지 배선 필요 *)
(* Rung L532 *)
%ML310.19 := NOT (%QX1.6.0 AND NOT %IX1.3.7 AND NOT %IX2.3.43 AND NOT %ML310.20) OR (%ML310.19 AND NOT %ML1.4 AND NOT %IX1.1.17);

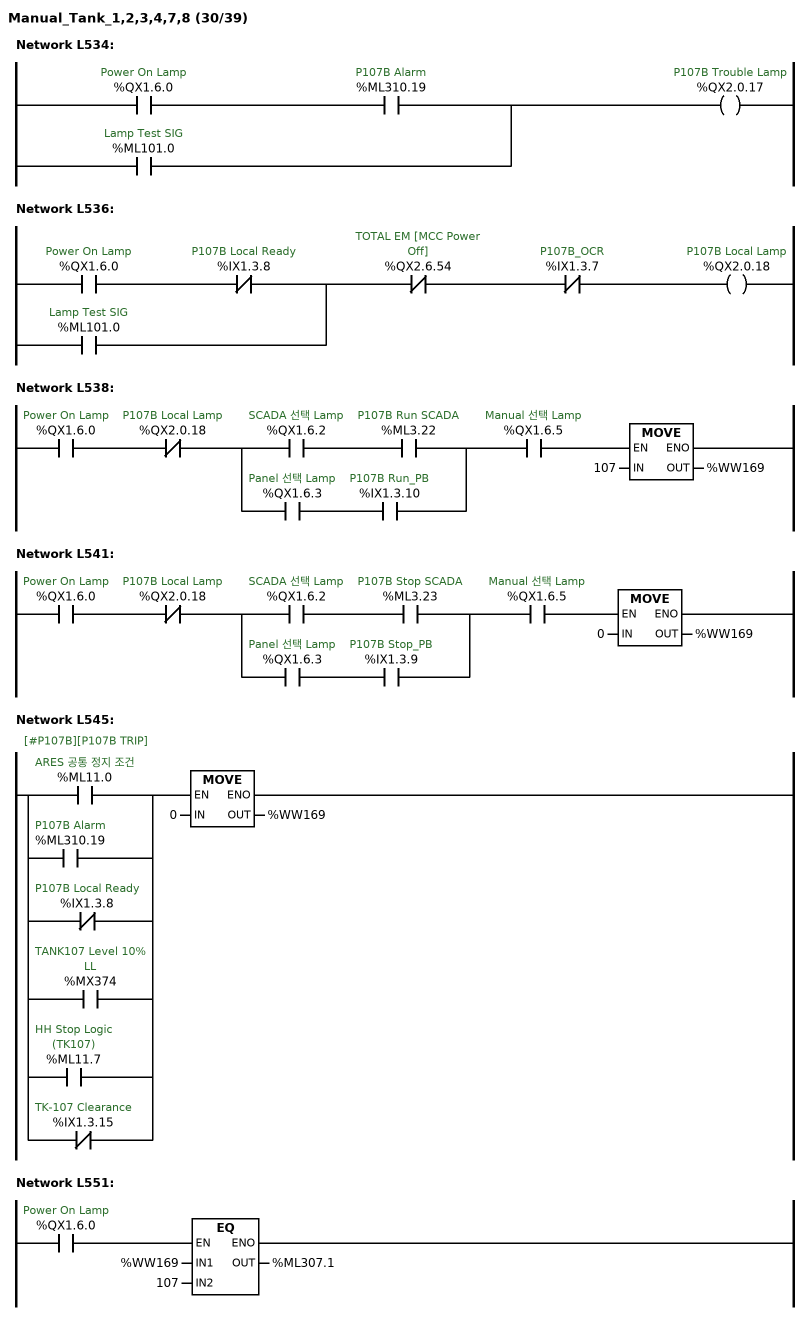
(* Rung L534 *)
%QX2.0.17 := (%QX1.6.0 AND %ML310.19) OR %ML101.0;
(* Rung L536 *)
%QX2.0.18 := ((%QX1.6.0 AND NOT %IX1.3.8) OR %ML101.0) AND NOT %QX2.6.54 AND NOT %IX1.3.7;
(* Rung L538 *)
IF %QX1.6.0 AND NOT %QX2.0.18 AND ((%QX1.6.2 AND %ML3.22) OR (%QX1.6.3 AND %IX1.3.10)) AND %QX1.6.5 THEN
    %WW169 := 107;
END_IF;
(* Rung L541 *)
IF %QX1.6.0 AND NOT %QX2.0.18 AND ((%QX1.6.2 AND %ML3.23) OR (%QX1.6.3 AND %IX1.3.9)) AND %QX1.6.5 THEN
    %WW169 := 0;
END_IF;
(* [#P107B][P107B TRIP] *)
(* Rung L545 *)
IF %ML11.0 OR %ML310.19 OR NOT %IX1.3.8 OR %MX374 OR %ML11.7 OR NOT %IX1.3.15 THEN %WW169 := 0; END_IF;
(* Rung L551 *)
IF %QX1.6.0 THEN %ML307.1 := %WW169 = 107; END_IF;

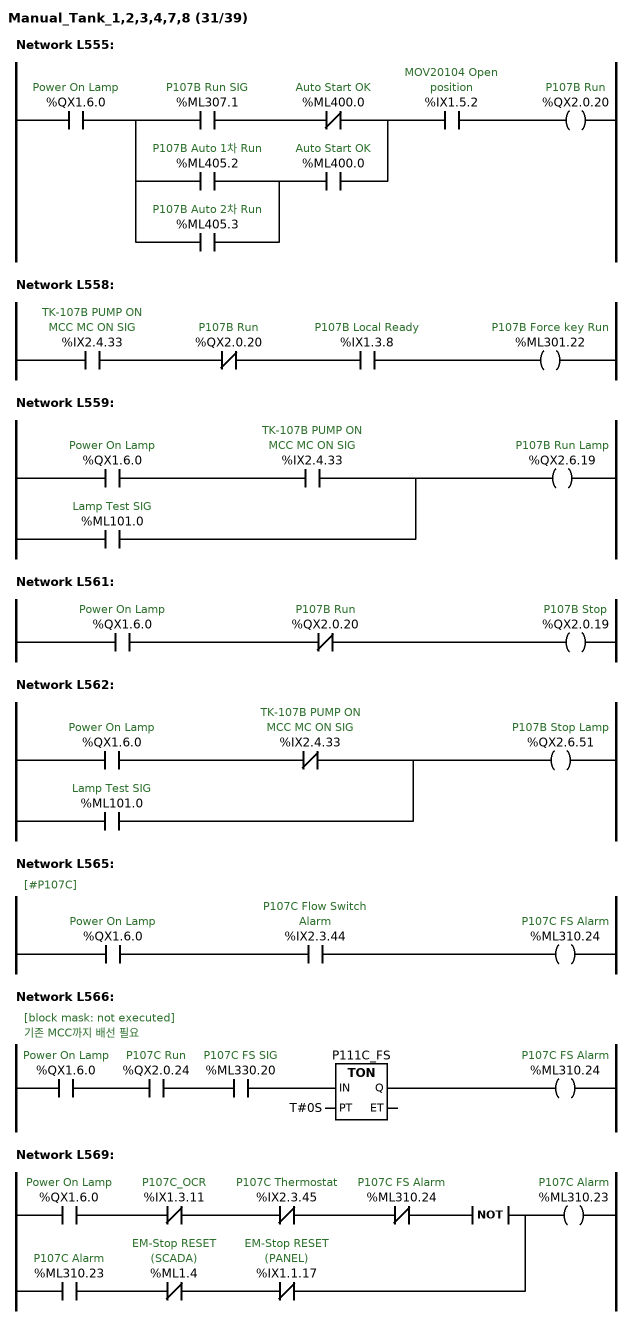
(* Rung L555 *)
%QX2.0.20 := %QX1.6.0 AND ((%ML307.1 AND NOT %ML400.0) OR ((%ML405.2 OR %ML405.3) AND %ML400.0)) AND %IX1.5.2;
(* Rung L558 *)
%ML301.22 := %IX2.4.33 AND NOT %QX2.0.20 AND %IX1.3.8;
(* Rung L559 *)
%QX2.6.19 := (%QX1.6.0 AND %IX2.4.33) OR %ML101.0;
(* Rung L561 *)
%QX2.0.19 := %QX1.6.0 AND NOT %QX2.0.20;
(* Rung L562 *)
%QX2.6.51 := (%QX1.6.0 AND NOT %IX2.4.33) OR %ML101.0;
(* [#P107C] *)
(* Rung L565 *)
%ML310.24 := %QX1.6.0 AND %IX2.3.44;
(* Rung L566 is block-masked: not executed *)
// P111C_FS(IN := %QX1.6.0 AND %QX2.0.24 AND %ML330.20, PT := T#0S);
// %ML310.24 := P111C_FS.Q;
(* 기존 MCC까지 배선 필요 *)
(* Rung L569 *)
%ML310.23 := NOT (%QX1.6.0 AND NOT %IX1.3.11 AND NOT %IX2.3.45 AND NOT %ML310.24) OR (%ML310.23 AND NOT %ML1.4 AND NOT %IX1.1.17);

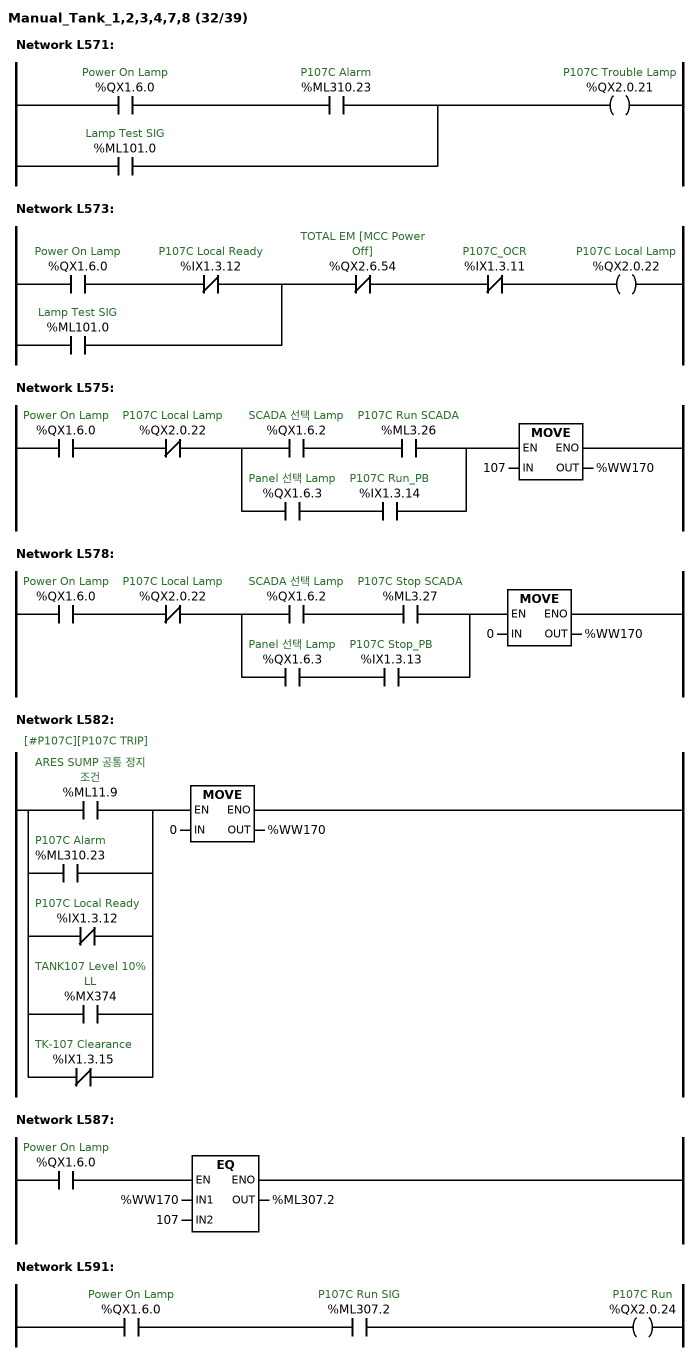
(* Rung L571 *)
%QX2.0.21 := (%QX1.6.0 AND %ML310.23) OR %ML101.0;
(* Rung L573 *)
%QX2.0.22 := ((%QX1.6.0 AND NOT %IX1.3.12) OR %ML101.0) AND NOT %QX2.6.54 AND NOT %IX1.3.11;
(* Rung L575 *)
IF %QX1.6.0 AND NOT %QX2.0.22 AND ((%QX1.6.2 AND %ML3.26) OR (%QX1.6.3 AND %IX1.3.14)) THEN
    %WW170 := 107;
END_IF;
(* Rung L578 *)
IF %QX1.6.0 AND NOT %QX2.0.22 AND ((%QX1.6.2 AND %ML3.27) OR (%QX1.6.3 AND %IX1.3.13)) THEN
    %WW170 := 0;
END_IF;
(* [#P107C][P107C TRIP] *)
(* Rung L582 *)
IF %ML11.9 OR %ML310.23 OR NOT %IX1.3.12 OR %MX374 OR NOT %IX1.3.15 THEN %WW170 := 0; END_IF;
(* Rung L587 *)
IF %QX1.6.0 THEN %ML307.2 := %WW170 = 107; END_IF;
(* Rung L591 *)
%QX2.0.24 := %QX1.6.0 AND %ML307.2;

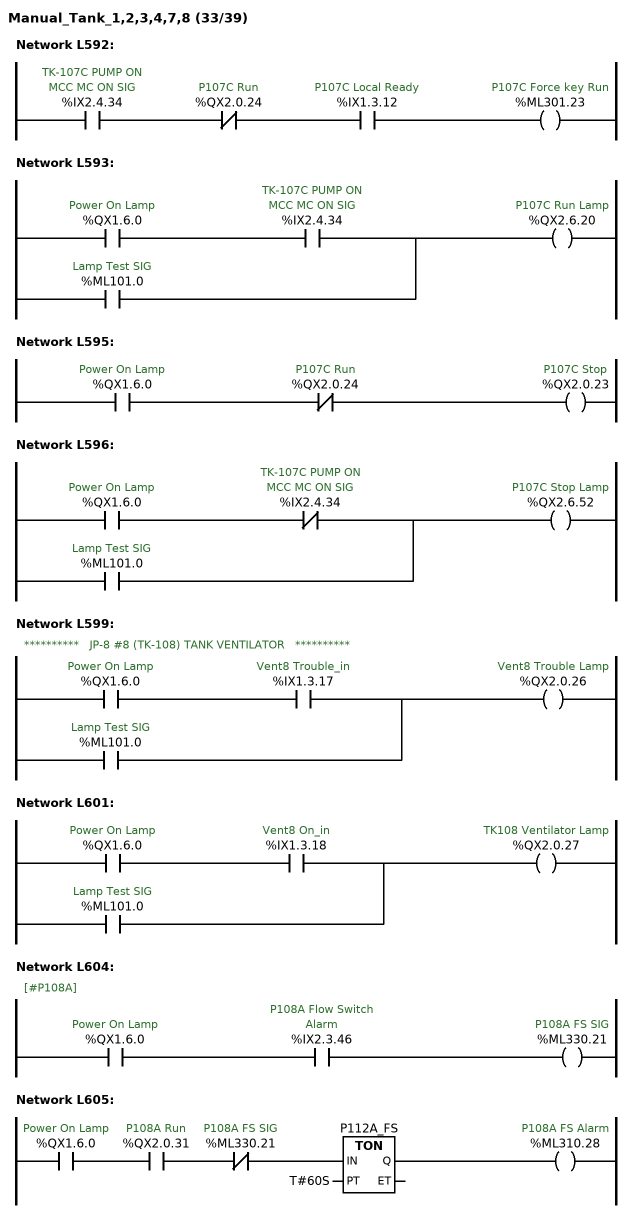
(* Rung L592 *)
%ML301.23 := %IX2.4.34 AND NOT %QX2.0.24 AND %IX1.3.12;
(* Rung L593 *)
%QX2.6.20 := (%QX1.6.0 AND %IX2.4.34) OR %ML101.0;
(* Rung L595 *)
%QX2.0.23 := %QX1.6.0 AND NOT %QX2.0.24;
(* Rung L596 *)
%QX2.6.52 := (%QX1.6.0 AND NOT %IX2.4.34) OR %ML101.0;
(* **********   JP-8 #8 (TK-108) TANK VENTILATOR   ********** *)
(* Rung L599 *)
%QX2.0.26 := (%QX1.6.0 AND %IX1.3.17) OR %ML101.0;
(* Rung L601 *)
%QX2.0.27 := (%QX1.6.0 AND %IX1.3.18) OR %ML101.0;
(* [#P108A] *)
(* Rung L604 *)
%ML330.21 := %QX1.6.0 AND %IX2.3.46;
(* Rung L605 *)
P112A_FS(IN := %QX1.6.0 AND %QX2.0.31 AND NOT %ML330.21, PT := T#60S);
%ML310.28 := P112A_FS.Q;

